FUNCTION_BLOCK FB_SkillHandler
VAR_INPUT
END_VAR
VAR_OUTPUT
END_VAR
VAR
	activSkill: POINTER TO FB_SKILL;
	_finished: BOOL;
END_VAR

IF activSkill^.bDone THEN
	_finished:=True;
END_IF

METHOD AbortActifSkill : BOOL
VAR_INPUT
END_VAR
activSkill^.M_Stop();
END_METHOD

PROPERTY ActiveSkillFinished : BOOL
GET
ActiveSkillFinished := _finished;
END_GET
END_PROPERTY

METHOD CallSkill : BOOL
VAR_INPUT
	pSkill : POINTER TO FB_SKILL;
END_VAR
activSkill:= pSkill;

//TODO Checks

pSkill^.M_Start();
END_METHOD

PROPERTY GetActivSkill : POINTER TO FB_SKILL
GET
GetActivSkill := activSkill;
END_GET
END_PROPERTY

END_FUNCTION_BLOCK

(* stored: Version 1.1.0.1, ProductVersion 3.1.4026.18
   POU FB_SkillHandler: Id {d564b0b9-96bf-4626-9d61-904bd7d86173}, SpecialFunc None
   Method AbortActifSkill: Id {10338084-d473-478a-aa27-fc35b9873599}
   Property ActiveSkillFinished: Id {e768b71e-2b8c-4823-b6e5-97c90ef183b8}
   Get Get: Id {8bd5e583-c1a7-40cf-800c-cc46c8f2112d}
   Method CallSkill: Id {d8fc5668-9fa7-43c2-a944-aada2bd4cb8c}
   Property GetActivSkill: Id {a76ffee6-6586-41ec-827c-b1a5d3fc1e96}
   Get Get: Id {d373d262-644a-4298-ae86-7673cc4dcfd7} *)
